FUNCTION_BLOCK PUBLIC EcMasterFrameStats IMPLEMENTS IEcTask
VAR_INPUT
END_VAR
VAR_OUTPUT
END_VAR
VAR
	iState : INT;
	masterFrameStats : Tc2_EtherCAT.FB_EcMasterFrameStatistic;
	_execute: BOOL;
	_done: BOOL;
	_busy: BOOL;
	_error: BOOL;
	_netId: AMSNETID;
END_VAR

CASE iState OF
	0:
		IF _execute THEN
			_done := FALSE;
			_busy := TRUE;
			_error := FALSE;
			masterFrameStats.bExecute := TRUE;
			IF masterFrameStats.bBusy THEN
				iState := 10;
				_execute := false;
			END_IF
		END_IF
	10:
		IF NOT masterFrameStats.bBusy THEN
			IF NOT masterFrameStats.bError THEN
				_done := TRUE;
			ELSE
				_error := TRUE;
			END_IF
			_busy := FALSE;
			masterFrameStats.bExecute := FALSE;
			iState := 0;
		END_IF
END_CASE

masterFrameStats(sNetId := Tc2_System.F_CreateAmsNetId(nIds := NetId));

{warning 'add method implementation '}
METHOD Abort : BOOL
masterFrameStats.bExecute := FALSE;
_busy := FALSE;
_execute := FALSE;
Abort := TRUE;
iState := 0;
END_METHOD

{warning 'add property implementation'}
PROPERTY Busy : BOOL
GET
Busy := _busy;
END_GET
END_PROPERTY

{warning 'add property implementation'}
PROPERTY Done : BOOL
GET
Done := _done;
END_GET
END_PROPERTY

{warning 'add property implementation'}
PROPERTY Error : BOOL
GET
Error := _error;
END_GET
END_PROPERTY

METHOD Execute : BOOL
VAR_INPUT
END_VAR
IF NOT Busy THEN
	Execute := _execute := TRUE;
END_IF
END_METHOD

PROPERTY FramesPerSecond  : LREAL
GET
FramesPerSecond := masterFrameStats.fFramesPerSecond;
END_GET
END_PROPERTY

PROPERTY LostFrames : UDINT
GET
LostFrames := masterFrameStats.nLostFrames;
END_GET
END_PROPERTY

PROPERTY LostQueuedFrames : udint
GET
LostQueuedFrames := masterFrameStats.nLostQueuedFrames;
END_GET
END_PROPERTY

{warning 'add property implementation'}
PROPERTY NetID : amsnetid
GET
NetID := _netId;
END_GET
SET
_netId := NetID;
END_SET
END_PROPERTY

PROPERTY QueuedFramesPerSecond : lreal
GET
QueuedFramesPerSecond := masterFrameStats.fQueuedFramesPerSecond;
END_GET
END_PROPERTY

END_FUNCTION_BLOCK

(* stored: Version 1.1.0.1, ProductVersion 3.1.4024.11
   POU EcMasterFrameStats: Id {33dd9519-af82-4727-b960-6626d65dc0c6}, SpecialFunc None
   Method Abort: Id {e556f6b8-e02b-4e4e-9e66-0f33545fa773}
   Property Busy: Id {4933a9cf-afb4-4849-9667-bb56a33baa20}
   Get Get: Id {4949444f-7eb7-4eda-a1ed-a3147feaabaa}
   Property Done: Id {f027a1a1-c8a2-45e0-bc3e-d2bf114bea68}
   Get Get: Id {39ad4e73-b75e-4c06-b436-9ea50d317907}
   Property Error: Id {38afbcaf-09a6-4590-a998-6697c99af61f}
   Get Get: Id {e72cb826-066b-49b9-867e-534f04380d83}
   Method Execute: Id {044b952a-f1c7-4d3f-897e-2e459fc6f9d4}
   Property FramesPerSecond: Id {f20a1475-9d98-4367-b1a5-1680b8f40c99}
   Get Get: Id {dd331882-f5cb-4f67-ba01-63ef26f8d70f}
   Property LostFrames: Id {aa4ec9bf-5814-4c12-9a96-654a7154817a}
   Get Get: Id {39ba628b-00c0-4875-ad7e-b01bce4b4a1c}
   Property LostQueuedFrames: Id {e6442b79-daa7-4d36-9c9a-5f8809366181}
   Get Get: Id {aa5c85a4-cf54-40f6-84be-24f49f0cee65}
   Property NetID: Id {e7bcc9df-3f40-4b03-8e16-d42eefbcda85}
   Get Get: Id {ba8442ba-238c-496e-aa18-c07eea232980}
   Set Set: Id {80212ed6-4b43-4ad0-b57a-6a0a019934ff}
   Property QueuedFramesPerSecond: Id {e864d0bb-5e97-43cc-9ae4-e1a9a82f4265}
   Get Get: Id {28bc28b0-80ce-4252-aa5b-b88991487f5c} *)
